// TIA Portal project "实验一_V20" (V20)

(* hardware
DEVICE "S7-300/ET200M station_1"  S7-300 station
   slot 0: "导轨_0"  Rail  6ES7 390-1***0-0AA0
   slot 2: "PLC_1"  CPU 314C-2 DP  6ES7 314-6CH04-0AB0  V3.3
      slot 0: "MPI 接口_1"  MPI
      slot 1: "DP 接口_1"  DP
      slot 2: "DI 24/DO 16_1"  DI24/DO16
      slot 3: "AI 5/AO 2_1"  AI5/AO2
      slot 4: "计数_1"  Counter
      slot 5: "定位_1"  Positioning
DEVICE "HMI_1"  KTP400 Comfort
   slot 0: "HMI_1"  KTP400 Comfort  6AV2 124-2DC01-0AX0  17.0.0.0
   slot 1: "HMI_RT_1"  KTP400 Comfort  6AV2 124-2DC01-0AX0  17.0.0.0
   slot 5: "HMI_1.IE_CP_1"  PROFINET Interface  17.0.0.0
      slot 1: "PROFINET Interface_1"  PROFINET Interface
         slot 1: "Port_1"  Port
   slot 7: "HMI_1.MPI/DP_CP_1"  MPI/DP Interface  17.0.0.0
*)

// ===== PLC "PLC_1"  CPU 314C-2 DP =====

VAR_GLOBAL   // PLC tag table "默认变量表"
   "启动按钮" AT %I0.0 : Bool;
   "停止按钮" AT %M10.0 : Bool;
   "运行状态" AT %M10.1 : Bool;
   "a" AT %Q5.0 : Bool;
   "b" AT %Q4.1 : Bool;
   "c" AT %Q4.2 : Bool;
   "d" AT %Q4.3 : Bool;
   "e" AT %Q4.4 : Bool;
   "f" AT %Q4.5 : Bool;
   "g" AT %Q4.6 : Bool;
   "h" AT %Q4.7 : Bool;
   "0.5Hz时钟" AT %M10.2 : Bool;
   "显示字符" AT %MW20 : Int;
   "时钟沿" AT %M10.3 : Bool;
   "Tag_1" AT %Q5.3 : Bool;
   "Tag_2" AT %Q5.2 : Bool;
   "Tag_3" AT %QB4 : Byte;
   "Tag_4" AT %QB5 : Byte;
END_VAR

DATA_BLOCK "LED显示模块_DB"   // DB1
{ S7_Optimized_Access := 'FALSE' }
VERSION : 0.1
// stored: InstanceOfName LED显示模块
"LED显示模块"
BEGIN
END_DATA_BLOCK

FUNCTION_BLOCK "LED显示模块"   // FB1, SCL
{ S7_Optimized_Access := 'FALSE' }
VERSION : 0.1
   VAR_INPUT
      显示字符 : Int;   // 10为A、11为b、12为C、13为d、14为E、15为F
   END_VAR
   VAR_OUTPUT
      "a" : Bool;
      "b" : Bool;
      c : Bool;
      d : Bool;
      "e" : Bool;
      f : Bool;
      g : Bool;
      h : Bool;
   END_VAR
BEGIN
   IF #显示字符=0 THEN//0字符显示
       #a := 1;
       #b := 1;
       #c := 1;
       #d := 1;
       #e := 1;
       #f := 1;
       #g := 0;
       #h := 1;
   END_IF;

   IF #显示字符 = 1 THEN//1字符显示
       #a := 0;
       #b := 1;
       #c := 1;
       #d := 0;
       #e := 0;
       #f := 0;
       #g := 0;
       #h := 1;
   END_IF;

   IF #显示字符 = 2 THEN//2字符显示
       #a := 1;
       #b := 1;
       #c := 0;
       #d := 1;
       #e := 1;
       #f := 0;
       #g := 1;
       #h := 1;
   END_IF;

   IF #显示字符 = 3 THEN//3字符显示
       #a := 1;
       #b := 1;
       #c := 1;
       #d := 1;
       #e := 0;
       #f := 0;
       #g := 1;
       #h := 1;
   END_IF;

   IF #显示字符 = 4 THEN//4字符显示
       #a := 0;
       #b := 1;
       #c := 1;
       #d := 0;
       #e := 0;
       #f := 1;
       #g := 1;
       #h := 1;
   END_IF;

   IF #显示字符 = 5 THEN//5字符显示
       #a := 1;
       #b := 0;
       #c := 1;
       #d := 1;
       #e := 0;
       #f := 1;
       #g := 1;
       #h := 1;
   END_IF;

   IF #显示字符 = 6 THEN//6字符显示
       #a := 1;
       #b := 0;
       #c := 1;
       #d := 1;
       #e := 1;
       #f := 1;
       #g := 1;
       #h := 1;
   END_IF;

   IF #显示字符 = 7 THEN//7字符显示
       #a := 1;
       #b := 1;
       #c := 1;
       #d := 0;
       #e := 0;
       #f := 0;
       #g := 0;
       #h := 1;
   END_IF;

   IF #显示字符 = 8 THEN//8字符显示
       #a := 1;
       #b := 1;
       #c := 1;
       #d := 1;
       #e := 1;
       #f := 1;
       #g := 1;
       #h := 1;
   END_IF;

   IF #显示字符 = 9 THEN//9字符显示
       #a := 1;
       #b := 1;
       #c := 1;
       #d := 1;
       #e := 0;
       #f := 1;
       #g := 1;
       #h := 1;
   END_IF;

   IF #显示字符 = 10 THEN//A字符显示
       #a := 1;
       #b := 1;
       #c := 1;
       #d := 0;
       #e := 1;
       #f := 1;
       #g := 1;
       #h := 1;
   END_IF;

   IF #显示字符 = 11 THEN//b字符显示
       #a := 0;
       #b := 0;
       #c := 1;
       #d := 1;
       #e := 1;
       #f := 1;
       #g := 1;
       #h := 1;
   END_IF;

   IF #显示字符 = 12 THEN//C字符显示
       #a := 1;
       #b := 0;
       #c := 0;
       #d := 1;
       #e := 1;
       #f := 1;
       #g := 0;
       #h := 1;
   END_IF;

   IF #显示字符 = 13 THEN//d字符显示
       #a := 0;
       #b := 1;
       #c := 1;
       #d := 1;
       #e := 1;
       #f := 0;
       #g := 1;
       #h := 1;
   END_IF;

   IF #显示字符 = 14 THEN//E字符显示
       #a := 1;
       #b := 0;
       #c := 0;
       #d := 1;
       #e := 1;
       #f := 1;
       #g := 1;
       #h := 1;
   END_IF;

   IF #显示字符 = 15 THEN//F字符显示
       #a := 1;
       #b := 0;
       #c := 0;
       #d := 0;
       #e := 1;
       #f := 1;
       #g := 1;
       #h := 1;
   END_IF;
END_FUNCTION_BLOCK

ORGANIZATION_BLOCK "Main"   // OB1, LAD
TITLE = "Main Program Sweep (Cycle)"
{ S7_Optimized_Access := 'FALSE' }
VERSION : 0.1
   VAR_TEMP
      OB1_EV_CLASS : Byte;   // Bits 0-3 = 1 (Coming event), Bits 4-7 = 1 (Event class 1)
      OB1_SCAN_1 : Byte;   // 1 (Cold restart scan 1 of OB 1), 3 (Scan 2-n of OB 1)
      OB1_PRIORITY : Byte;   // Priority of OB Execution
      OB1_OB_NUMBR : Byte;   // 1 (Organization block 1, OB1)
      OB1_RESERVED_1 : Byte;   // Reserved for system
      OB1_RESERVED_2 : Byte;   // Reserved for system
      OB1_PREV_CYCLE : Int;   // Cycle time of previous OB1 scan (milliseconds)
      OB1_MIN_CYCLE : Int;   // Minimum cycle time of OB1 (milliseconds)
      OB1_MAX_CYCLE : Int;   // Maximum cycle time of OB1 (milliseconds)
      OB1_DATE_TIME : Date_And_Time;   // Date and time OB1 started
   END_VAR
   VAR_TEMP   // added for the SCL form of the ladder/FBD networks
      _w1 : Bool;
   END_VAR
BEGIN

REGION Network 1: 运行状态定义
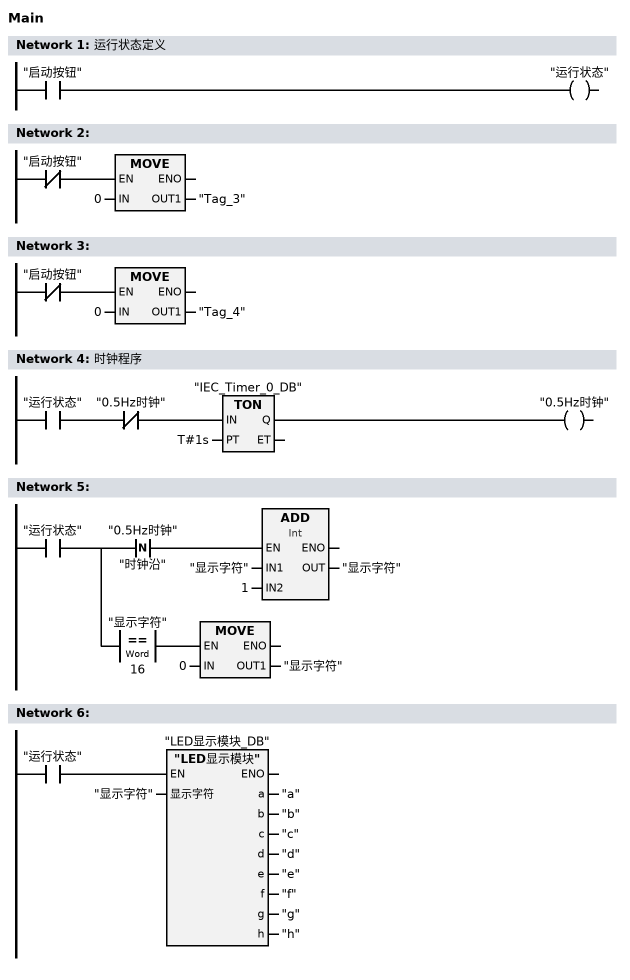
   RUNG wire#powerrail
      Contact( "启动按钮" )
      Coil( "运行状态" )
   END_RUNG
   // the same network as SCL:
   "运行状态" := "启动按钮";
END_REGION

REGION Network 2
   RUNG wire#powerrail
      I_Contact( "启动按钮" )
      { S7_GenerateENO := "TRUE" } Move(in := 0, out1 => "Tag_3")
   END_RUNG
   // the same network as SCL:
   IF NOT "启动按钮" THEN "Tag_3" := 0; END_IF;
END_REGION

REGION Network 3
   RUNG wire#powerrail
      I_Contact( "启动按钮" )
      { S7_GenerateENO := "TRUE" } Move(in := 0, out1 => "Tag_4")
   END_RUNG
   // the same network as SCL:
   IF NOT "启动按钮" THEN "Tag_4" := 0; END_IF;
END_REGION

REGION Network 4: 时钟程序
   "IEC_Timer_0_DB".TON(IN := "运行状态" AND NOT "0.5Hz时钟", PT := T#1s);
   "0.5Hz时钟" := "IEC_Timer_0_DB".Q;
END_REGION

REGION Network 5
   RUNG wire#powerrail
      Contact( "运行状态" )
      wire#w1
      N_Contact(operand := "0.5Hz时钟", bit := "时钟沿")
      { S7_Templates := "SrcType := Int"; S7_GenerateENO := "TRUE" } Add(in1 := "显示字符", in2 := 1, out => "显示字符")
   END_RUNG
   RUNG wire#w1
      { S7_Templates := "SrcType := Word" } EQ_Contact(in1 := "显示字符", in2 := 16)
      { S7_GenerateENO := "TRUE" } Move(in := 0, out1 => "显示字符")
   END_RUNG
   // the same network as SCL:
   #_w1 := "运行状态" AND NOT "0.5Hz时钟" AND "时钟沿";   // falling edge of "0.5Hz时钟"
   "时钟沿" := "0.5Hz时钟";
   IF #_w1 THEN "显示字符" := "显示字符" + 1; END_IF;
   IF "运行状态" AND ("显示字符" = 16) THEN "显示字符" := 0; END_IF;
END_REGION

REGION Network 6
   RUNG wire#powerrail
      Contact( "运行状态" )
      "LED显示模块_DB"(显示字符 := "显示字符", "a" => "a", "b" => "b", c => "c", d => "d", "e" => "e", f => "f", g => "g", h => "h")
   END_RUNG
   // the same network as SCL:
   IF "运行状态" THEN
       "LED显示模块_DB"(显示字符 := "显示字符",   // "LED显示模块"
                    "a" => "a",
                    "b" => "b",
                    c => "c",
                    d => "d",
                    "e" => "e",
                    f => "f",
                    g => "g",
                    h => "h");
   END_IF;
END_REGION
END_ORGANIZATION_BLOCK

(* ===== HMI "HMI_RT_1" =====
system functions are stored by id; their names below are inferred from use
connection "HMI_连接_1": IF1 B, SIMATIC S7 300/400 MPI

HMI tags "默认变量表"
   "Tag_ScreenNumber" : UInt, internal
   "a" : Bool = PLC a AT %Q5.0, 1 s
   "b" : Bool = PLC b AT %Q4.1, 1 s
   "c" : Bool = PLC c AT %Q4.2, 1 s
   "d" : Bool = PLC d AT %Q4.3, 1 s
   "e" : Bool = PLC e AT %Q4.4, 1 s
   "f" : Bool = PLC f AT %Q4.5, 1 s
   "g" : Bool = PLC g AT %Q4.6, 1 s
   "h" : Bool = PLC h AT %Q4.7, 1 s

screen "根画面" 480x212, template "模板_1"
   on GenerateScreen: SetTag("Tag_ScreenNumber", 1)
   Rectangle "矩形_1" at 216,8 size 56x8
      Appearance <- "a"
   Rectangle "矩形_2" at 272,16 size 8x56
      Appearance <- "b"
   Rectangle "矩形_3" at 272,80 size 8x56
      Appearance <- "c"
   Rectangle "矩形_4" at 216,136 size 56x8
      Appearance <- "d"
   Rectangle "矩形_5" at 216,72 size 56x8
      Appearance <- "g"
   Rectangle "矩形_6" at 208,16 size 8x56
      Appearance <- "f"
   Rectangle "矩形_7" at 208,80 size 8x56
      Appearance <- "e"
   Rectangle "矩形_8" at 296,136 size 8x8
      Appearance <- "h"

Template "模板_1" 480x212
   Button "退出" at 379,148 size 63x63; TextOff '退出'; PictureOff "ExitRuntime_KTP400_Comfort_TR"; PictureOn "ExitRuntime_KTP400_Comfort_TR"
      on Release: StopRuntime(0)
   Button "Template_Button" at 265,148 size 63x63; TextOff 'Text'
   Button "Template_Button_1" at 151,148 size 63x63; TextOff 'Text'
   Button "起始画面" at 37,148 size 63x63; TextOff '起始画面'; PictureOff "NavigateHome_KTP400_Comfort_TR"; PictureOn "NavigateHome_KTP400_Comfort_TR"
      on Release: ActivateScreen("根画面", 0)
*)